// TIA Portal V17 export
// export: Created 2024-06-14T09:53:45.5085394Z, ExportSetting WithDefaults, DisplayName Totally Integrated Automation Portal, DisplayVersion V17, DisplayName TIA Portal Openness, DisplayVersion V17, DisplayName TIA Portal Version Control Interface, DisplayVersion V17, DisplayName Simotion SCOUT TIA, DisplayVersion 5.4.3.0, DisplayName SINAMICS Startdrive Advanced, DisplayVersion V17 SP1 Update 1, DisplayName SINAMICS Startdrive G110M, G120, G120C, G120D, G120P, G115D, DisplayVersion V17 SP1 Update 1, DisplayName SINAMICS Startdrive G130, G150, S120, S150, SINAMICS MV, S210, DisplayVersion V17 SP1 Update 1, DisplayName STEP 7 Professional, DisplayVersion V17, DisplayName STEP 7 Safety, DisplayVersion V17, DisplayName WinCC Professional, DisplayVersion V17
VAR_GLOBAL   // PLC tag table "Default tag table"
   A_Tag_1 AT %M102.0 : Bool;
   A_Tag_2 AT %M102.1 : Bool;
   A_Tag_3 AT %M102.2 : Bool;
   A_Tag_4 AT %M102.3 : Bool;
   A_Tag_5 AT %M102.4 : Bool;
   Tag_1 AT %M200.0 : Bool;
   P_Trig08 AT %M2.0 : Bool;
   Tag_3 AT %M9.0 : Bool;
   Tag_4 AT %M9.1 : Bool;
   Tag_5 AT %M200.2 : Bool;
   A_Tag_11 AT %M2.1 : Bool;
   Tag_6 AT %M200.1 : Bool;
   Tag_7 AT %M110.0 : Bool;
   Tag_8 AT %M210.0 : Bool;
   Tag_9 AT %M210.1 : Bool;
   Tag_10 AT %M210.2 : Bool;
   Tag_11 AT %M210.4 : Bool;
   Tag_12 AT %M210.5 : Bool;
   Tag_13 AT %M210.6 : Bool;
   temp AT %M300.0 : Bool;
   Tag_14 AT %M210.7 : Bool;
   Tag_15 AT %M9.2 : Bool;
   Tag_17 AT %MW13 : Int;
   Tag_18 AT %MW15 : Int;
   Master1_Done_Bit AT %M11.0 : Bool;
   Master_Error_Bit AT %M11.1 : Bool;
   Tag_19 AT %MW500 : Word;
   Tag_20 AT %MW100 : Int;
   Tag_21 AT %M9.7 : Bool;
   Tag_22 AT %M20.0 : Bool;
   Tag_23 AT %M20.1 : Bool;
   Tag_24 AT %M22.0 : Bool;
   Tag_25 AT %M22.1 : Bool;
   System_Byte AT %MB1 : Byte;
   FirstScan AT %M1.0 : Bool;
   DiagStatusUpdate AT %M1.1 : Bool;
   AlwaysTRUE AT %M1.2 : Bool;
   AlwaysFALSE AT %M1.3 : Bool;
   Clock_Byte AT %MB0 : Byte;
   Clock_10Hz AT %M0.0 : Bool;
   Clock_5Hz AT %M0.1 : Bool;
   "Clock_2.5Hz" AT %M0.2 : Bool;
   Clock_2Hz AT %M0.3 : Bool;
   "Clock_1.25Hz" AT %M0.4 : Bool;
   Clock_1Hz AT %M0.5 : Bool;
   "Clock_0.625Hz" AT %M0.6 : Bool;
   "Clock_0.5Hz" AT %M0.7 : Bool;
   Tag_26 AT %M503.6 : Bool;
   Tag_27 AT %M23.0 : Bool;
   Tag_28 AT %M25.0 : Bool;
   Tag_29 AT %M25.1 : Bool;
   Tag_30 AT %M26.0 : Bool;
   Tag_31 AT %M27.0 : Bool;
   Tag_32 AT %M27.1 : Bool;
   Tag_33 AT %M27.2 : Bool;
   Tag_34 AT %M27.3 : Bool;
   Tag_35 AT %M27.4 : Bool;
   Tag_36 AT %M27.5 : Bool;
   Tag_37 AT %M27.6 : Bool;
   Tag_38 AT %M27.7 : Bool;
   Tag_39 AT %M28.0 : Bool;
   Tag_40 AT %M28.1 : Bool;
   Tag_41 AT %M28.2 : Bool;
   Tag_42 AT %M28.3 : Bool;
   Tag_43 AT %M28.4 : Bool;
   Tag_44 AT %M28.5 : Bool;
   Tag_45 AT %M28.6 : Bool;
   Tag_2 AT %M211.0 : Bool;
   Tag_16 AT %M211.2 : Bool;
   Tag_46 AT %M211.3 : Bool;
   Tag_47 AT %M212.0 : Bool;
   Tag_48 AT %M212.1 : Bool;
   Tag_49 AT %M212.2 : Bool;
   Tag_50 AT %M212.3 : Bool;
   Tag_51 AT %M212.4 : Bool;
   Tag_52 AT %M213.5 : Bool;
   Tag_53 AT %M212.5 : Bool;
   Tag_54 AT %M212.6 : Bool;
   Tag_55 AT %M212.7 : Bool;
   Tag_56 AT %M213.4 : Bool;
   Tag_57 AT %M213.0 : Bool;
   Tag_58 AT %M213.1 : Bool;
   Tag_59 AT %M213.2 : Bool;
   Tag_60 AT %M213.3 : Bool;
   Tag_61 AT %M214.0 : Bool;
   Tag_62 AT %M214.1 : Bool;
   Tag_63 AT %M214.2 : Bool;
   Tag_64 AT %M214.3 : Bool;
   Tag_65 AT %M214.4 : Bool;
   Tag_66 AT %M214.5 : Bool;
   Tag_67 AT %M214.6 : Bool;
   Tag_68 AT %MW1000 : Int;
   Tag_69 AT %M9.3 : Bool;
   Tag_70 AT %M214.7 : Bool;
   NUM_0 AT %I4.0 : Bool;
   NUM_1 AT %I4.1 : Bool;
   NUM_2 AT %I4.2 : Bool;
   NUM_3 AT %I4.3 : Bool;
   NUM_4 AT %I4.4 : Bool;
   NUM_5 AT %I4.5 : Bool;
   NUM_6 AT %I4.6 : Bool;
   NUM_7 AT %I4.7 : Bool;
   NUM_8 AT %I5.0 : Bool;
   NUM_9 AT %I5.1 : Bool;
   ENTER AT %I5.2 : Bool;
   Clear AT %I5.3 : Bool;
   Tag_71 AT %M2.2 : Bool;
   S5_SENSOR_CYL6 AT %I3.6 : Bool;
   S5_DOWN_CONVEYOR AT %I3.7 : Bool;
   SCREEN AT %I5.4 : Bool;
   BPCL_CY AT %I5.5 : Bool;
   MALABAR_GAS AT %I5.6 : Bool;
   "i5.7" AT %I5.7 : Bool;
   "q3.5" AT %Q3.5 : Bool;
   "q3.6" AT %Q3.6 : Bool;
   "q3.7" AT %Q3.7 : Bool;
   Tag_72 AT %M201.0 : Bool;
   Tag_73 AT %M201.1 : Bool;
   Tag_74 AT %M201.2 : Bool;
   Tag_75 AT %M99.7 : Bool;
   cylinder_pos AT %I2.4 : Bool;
   commercial AT %I2.5 : Bool;
   cylinder_exit AT %I2.6 : Bool;
   S5_CYCLE_START_L2 AT %I0.2 : Bool;
   S5_CYCLE_RESET_L2 AT %I0.3 : Bool;
   SEQ_RESET AT %I0.4 : Bool;
   MANUAL_SEQ AT %I0.5 : Bool;
   "i0.6" AT %I0.6 : Bool;
   "i0.7" AT %I0.7 : Bool;
   SEQ_RESET_L2 AT %I2.7 : Bool;
   S5_STOPPER_SENSOR AT %I3.0 : Bool;
   S5_SENSOR_CYL1 AT %I3.1 : Bool;
   S5_SENSOR_CYL2 AT %I3.2 : Bool;
   S5_SENSOR_CYL3 AT %I3.3 : Bool;
   S5_SENSOR_CYL4 AT %I3.4 : Bool;
   S5_SENSOR_CYL5 AT %I3.5 : Bool;
   DIVERTER AT %Q1.4 : Bool;
   PLC_LIVE AT %Q1.5 : Bool;
   spare_2 AT %Q1.6 : Bool;
   spare_3 AT %Q1.7 : Bool;
   S5_STOPPER_OP AT %Q2.0 : Bool;
   S5_LIFT_CYL6 AT %Q2.1 : Bool;
   S5_LIFT_CYL5 AT %Q2.2 : Bool;
   stopper AT %Q0.0 : Bool;
   Tag_76 AT %M888.7 : Bool;
   Tag_77 AT %M888.5 : Bool;
   Tag_78 AT %M888.6 : Bool;
   Seq_Lifttable_done AT %M100.7 : Bool;
   entry_data AT %MW90 : Int;
   MC_Reset AT %M100.2 : Bool;
   Tag_79 AT %M100.4 : Bool;
   "anti jammer" AT %M100.5 : Bool;
   Tag_80 AT %M100.6 : Bool;
   Tag_81 AT %M202.0 : Bool;
   Tag_82 AT %M202.1 : Bool;
   Tag_83 AT %M202.2 : Bool;
   Tag_84 AT %M202.4 : Bool;
   Tag_85 AT %M202.5 : Bool;
   Tag_86 AT %M202.6 : Bool;
   Tag_87 AT %M202.7 : Bool;
   Tag_88 AT %M203.0 : Bool;
   Tag_89 AT %M203.2 : Bool;
   Tag_90 AT %M203.1 : Bool;
   Tag_91 AT %M203.5 : Bool;
   Tag_92 AT %M203.7 : Bool;
   Tag_93 AT %M204.0 : Bool;
   Tag_94 AT %M204.1 : Bool;
   Tag_95 AT %M204.2 : Bool;
   Tag_96 AT %M204.3 : Bool;
   Tag_97 AT %M204.6 : Bool;
   Tag_98 AT %M203.4 : Bool;
   Tag_99 AT %M999.7 : Bool;
   Tag_101 AT %M5.7 : Bool;
   Tag_103 AT %M5.6 : Bool;
   Tag_104 AT %M500.0 : Bool;
   Tag_105 AT %M700.0 : Bool;
   Tag_106 AT %M700.1 : Bool;
   Check_Stopper AT %I6.0 : Bool;
   Check_presence AT %I6.1 : Bool;
   Check_pusher AT %I6.2 : Bool;
   Check_antijammer AT %I6.3 : Bool;
   Check_start_PB AT %I6.4 : Bool;
   Check_reset_PB AT %I6.5 : Bool;
   Check_Down_line_jammer AT %I6.6 : Bool;
   Correction_Stopper_sensor AT %I6.7 : Bool;
   Correction_Lift_sensor AT %I7.0 : Bool;
   Correction_Jammer_sensor AT %I7.1 : Bool;
   Correction_Start_PB AT %I7.2 : Bool;
   Correction_Reset_PB AT %I7.3 : Bool;
   Check_stopper_op AT %Q4.0 : Bool;
   Check_lift_table AT %Q4.1 : Bool;
   Check_pusher_op AT %Q4.2 : Bool;
   Correction_Stopper_solenoid AT %Q4.3 : Bool;
   Correction_Lift_solenoid AT %Q4.4 : Bool;
END_VAR
